INTERFACE I_VisionMode_StatusOnly EXTENDS __SYSTEM.IQueryInterface

{attribute 'monitoring' := 'call'}
// Name or description of this mode
PROPERTY Name : STRING
GET
END_GET
END_PROPERTY

END_INTERFACE

(* stored: Version 1.1.0.1, ProductVersion 3.1.4024.12
   Itf I_VisionMode_StatusOnly: Id {d39b5128-c8a6-4334-85c6-fc07f8fa9e11}
   Property Name: Id {783f4089-51e2-4fec-b6d9-b0e373fa969c}
   Get Get: Id {d634363b-13be-4432-9a3f-f15de60392d9} *)
